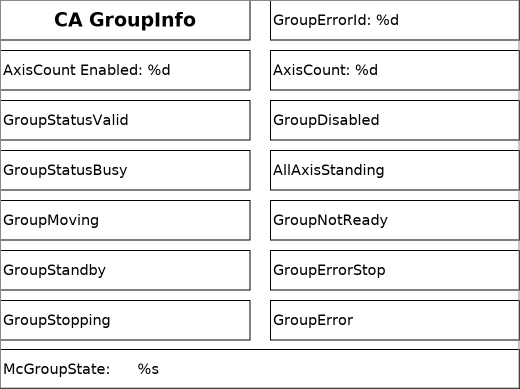
VISUALIZATION GROUP_VISU  // 520x389
VAR_IN_OUT
	stGroupInfo   : ST_GROUP_INFO;
  sGroupState   : string(60);
END_VAR
    Rectangle (0,100 250x40), "GroupStatusValid", colour toggle: stGroupInfo.GroupStatusValid
    Rectangle (0,150 250x40), "GroupStatusBusy", colour toggle: stGroupInfo.GroupStatusBusy
    Rectangle (0,200 250x40), "GroupMoving", colour toggle: stGroupInfo.GroupMoving
    Rectangle (270,250 250x40), "GroupErrorStop", colour toggle: stGroupInfo.GroupErrorStop
    Rectangle (270,200 250x40), "GroupNotReady", colour toggle: stGroupInfo.GroupNotReady
    Rectangle (0,250 250x40), "GroupStandby", colour toggle: stGroupInfo.GroupStandby
    Rectangle (0,300 250x40), "GroupStopping", colour toggle: stGroupInfo.GroupStopping
    Rectangle (270,100 250x40), "GroupDisabled", colour toggle: stGroupInfo.GroupDisabled
    Rectangle (270,150 250x40), "AllAxisStanding", colour toggle: stGroupInfo.AllAxesStanding
    Rectangle (270,300 250x40), "GroupError", colour toggle: stGroupInfo.GroupError
    Rectangle (270,0 250x40), "GroupErrorId: %d", text variable: stGroupInfo.GroupErrorId
    Rectangle (270,50 250x40), "AxisCount: %d", text variable: stGroupInfo.AxisCount
    Rectangle (0,349 520x40), "McGroupState: %s", text variable: sGroupState
    Rectangle (0,0 250x40), "CA GroupInfo"
    Rectangle (0,50 250x40), "AxisCount Enabled: %d", text variable: stGroupInfo.AxisCountEnabled
END_VISUALIZATION

(* stored: Version 1.1.0.1
   Visu GROUP_VISU: Id {f3d551c7-1cd0-498d-b8ce-ece3e2b79f70} *)
